INTERFACE ITF_EM_Check_Weigher

END_INTERFACE

(* stored: Version 1.1.0.1, ProductVersion 3.1.4024.12
   Itf ITF_EM_Check_Weigher: Id {1cdd2504-f1c5-48a2-88af-449a0b20e71e} *)
